FUNCTION_BLOCK FB3_HmiTF1800_UserlevelManagement
VAR_INPUT
	
	bLoginPB 					: BOOL;
	bLogoutPB 					: BOOL;
	iLoginNameId 				: REFERENCE TO INT; // The LoginName selection in HMI during User Login Pop-up Screen, the choosen user will translated as Array ID No and pass here.
	sPasswordField 				: REFERENCE TO STRING; // Similar to Var In/Out so that i can clear the password if login failed
	
	iUM_SelectedLoginNameId	 	: REFERENCE TO INT;		// User Management - Selected Login Name ID (Array No)

	sUM_CurrentPassword			: REFERENCE TO STRING;	// User Management - Current Password (For password change only)
	sUM_NewPassword				: REFERENCE TO STRING;	// User Management - New Password (For password change or new user registration)
	sUM_ConfirmPassword			: REFERENCE TO STRING;	// User Management - New Password (For password change or new user registration)

	sUM_NewUserLoginName		: REFERENCE TO STRING;	// User Management - New User Login Name
	sUM_NewUserGroupId			: REFERENCE TO INT;		// User Management - Select from UserGroupList

	sUM_NewUserOperatorIdentifier	: REFERENCE TO STRING;
	sUM_NewUserActorType			: REFERENCE TO eActor;
	sUM_NewUserLastName				: REFERENCE TO STRING;
	sUM_NewUserFirstName			: REFERENCE TO STRING;
//	sUM_NewUserGroupName			: REFERENCE TO WSTRING; // Generated by reference eto sUM_NewUserGroupId
	
	bUM_CreatePB				: BOOL;		// User Management - Button for New User creation
	bUM_EditPB					: BOOL;		// User Management - Button for Edit User
	bUM_DeletePB				: BOOL;		// User Management - Button for Delete User
	bUM_EnablePB				: BOOL; 	// to Enable selected User
	bUM_DisablePB				: BOOL; 	// to Temporary Disable selected User
	bUM_ConfirmPB				: BOOL;		// for Edit, Delete and Disable used. click to save
	bUM_ReturnPB				: BOOL;		// for Edit, Delete and Disable used, click to return without save.
		
END_VAR
VAR_OUTPUT
	dsHmiUserStatus_Active		: DS_HmiUserStatus;
	dsHmiUserStatus_Login		: DS_HmiUserStatus;
	dsHmiUserStatus_Logout		: DS_HmiUserStatus;
	
//	iActiveUserGroupId			: INT;
//	sActiveLoginName			: STRING;
	
//	sActiveOperatorIdentifier	: STRING;
//	eActiveActorType			: eActor;
//	sActiveLastName				: STRING;
//	sActiveFirstName			: STRING;
	wsActiveUserGroupName		: WSTRING;
	sMessage					: STRING;
	
END_VAR
VAR
	tsLocalSystemTimeStruct		: TIMESTRUCT;
	dsHmiUserStatus_Empty		: DS_HmiUserStatus;

	ARsUserGroup 				: ARRAY [0..5] OF WSTRING;	// Default UserGroup - Must Matched with HMI UserGroup Naming
	
	bLoginPBRE		: R_TRIG;
	bLogoutPBRE		: R_TRIG;
	bUM_CreatePBRE	: R_TRIG;
	bUM_EditPBRE	: R_TRIG;
	bUM_DeletePBRE	: R_TRIG;
	bUM_DisablePBRE	: R_TRIG;
	iCase: INT;
	sMessageDelayTimer: TON;
	iFL: INT;
	bDuplicatedLoginName: BOOL;
	bDuplicatedOperatorId: BOOL;
	bUserDBMax: BOOL;
	iUserDBVacantField: INT;
	bUM_ConfirmPBRE: R_TRIG;
	bUM_ReturnPBRE: R_TRIG;
	btest: BOOL;
	bUM_EnablePBRE: R_TRIG;
	tLoginActivatedTimer: TON;
	tLogoutActivatedTimer: TON;
	ntGetTime: NT_GetTime;
	t1s: TON;
END_VAR
	
VAR PERSISTENT
	dsHmiUserReg 			: DS_HmiUserReg;
END_VAR

t1s(IN:=NOT t1s.Q , PT:=T#0.5S , Q=> , ET=> );

// Get System Time
ntGetTime(	NETID:='' , START:=t1s.Q , TMOUT:= T#5S, TIMESTR=> tsLocalSystemTimeStruct);

tsLocalSystemTimeStruct.wYear;
tsLocalSystemTimeStruct.wMonth;
tsLocalSystemTimeStruct.wDay;
tsLocalSystemTimeStruct.wHour;
tsLocalSystemTimeStruct.wMinute;
tsLocalSystemTimeStruct.wSecond;
tsLocalSystemTimeStruct.wMilliseconds;
tsLocalSystemTimeStruct.wDayOfWeek;


// Default UserGroup - Must Matched with HMI UserGroup Naming
ARsUserGroup[0]			:= 	STRING_TO_WSTRING('GUEST');
ARsUserGroup[1]			:= 	STRING_TO_WSTRING('OPERATOR');
ARsUserGroup[2]			:=	STRING_TO_WSTRING('TECHNICIAN');
ARsUserGroup[3]			:=	STRING_TO_WSTRING('ENGINEER');
ARsUserGroup[4]			:=	STRING_TO_WSTRING('ADMIN');
ARsUserGroup[5]			:=	STRING_TO_WSTRING('JKS');
//ARsUserGroup[6]			:=	STRING_TO_WSTRING('');
//ARsUserGroup[7]			:=	STRING_TO_WSTRING('');	

// Default SuperAdmin
dsHmiUserReg.ARbUserStatus[dsHmiUserReg.iQtyUserReg+1]			:= 	TRUE		;
dsHmiUserReg.AReActorType[dsHmiUserReg.iQtyUserReg+1]			:= 	0			; //Human
dsHmiUserReg.ARiUserGroupID[dsHmiUserReg.iQtyUserReg+1]			:= 	5			; //Highest level - JKS Admin
dsHmiUserReg.ARsFirstName[dsHmiUserReg.iQtyUserReg+1]			:= 	'Machine'	;
dsHmiUserReg.ARsLastName[dsHmiUserReg.iQtyUserReg+1]			:= 	'Maker'		;
dsHmiUserReg.ARsLoginName[dsHmiUserReg.iQtyUserReg+1]			:= 	'SoftwareManager'	;
dsHmiUserReg.ARsOperatorIdentifier[dsHmiUserReg.iQtyUserReg+1]	:= 	'Software Manager'	;
dsHmiUserReg.ARsPw[dsHmiUserReg.iQtyUserReg+1]					:= 	'7189'	;
dsHmiUserReg.ARwsUserGroupName[dsHmiUserReg.iQtyUserReg+1]		:= 	ARsUserGroup[5]	;


// R_TRIG
bLoginPBRE		(CLK:=bLoginPB , 		Q=> );
bLogoutPBRE		(CLK:=bLogoutPB , 		Q=> );

bUM_CreatePBRE	(CLK:=bUM_CreatePB , 	Q=> );
bUM_EditPBRE	(CLK:=bUM_EditPB , 		Q=> );
bUM_DeletePBRE	(CLK:=bUM_DeletePB , 	Q=> );
bUM_EnablePBRE	(CLK:=bUM_EnablePB , 	Q=> );
bUM_DisablePBRE	(CLK:=bUM_DisablePB , 	Q=> );
bUM_ConfirmPBRE	(CLK:=bUM_ConfirmPB , 	Q=> );
bUM_ReturnPBRE	(CLK:=bUM_ReturnPB , 	Q=> );


// Delay off
tLoginActivatedTimer(IN:=dsHmiUserStatus_Login.bActivatedFlag , PT:=T#1S , Q=> , ET=> );
IF tLoginActivatedTimer.Q THEN
	dsHmiUserStatus_Login.bActivatedFlag := FALSE;
END_IF

tLogoutActivatedTimer(IN:=dsHmiUserStatus_Logout.bActivatedFlag , PT:=T#1S , Q=> , ET=> );
IF tLogoutActivatedTimer.Q THEN
	dsHmiUserStatus_Logout.bActivatedFlag := FALSE;
END_IF



// Action 

	IF iCase = 0 THEN
		
		IF 	bLoginPBRE.Q AND iLoginNameId > 0 AND iLoginNameId <= dsHmiUserReg.iQtyUserReg +1 AND sPasswordField <> '' THEN
			iCase := 11; // Login 
			
		ELSIF bLogoutPBRE.Q THEN
			iCase := 21; //	Logout
			
		ELSIF bUM_CreatePBRE.Q AND dsHmiUserStatus_Login.sUserGroupId >= 4 THEN
			iCase := 31; //	User Management -> New User Creation
			
		ELSIF bUM_EditPBRE.Q AND dsHmiUserStatus_Login.sUserGroupId >= 4 AND iUM_SelectedLoginNameId > 0 AND iUM_SelectedLoginNameId <= dsHmiUserReg.iQtyUserReg +1 THEN
			iCase := 41; //	User Management -> Edit User
			
		ELSIF bUM_DeletePBRE.Q AND dsHmiUserStatus_Login.sUserGroupId >= 4 AND iUM_SelectedLoginNameId > 0 AND iUM_SelectedLoginNameId <= dsHmiUserReg.iQtyUserReg +1 
		AND dsHmiUserReg.ARsLoginName[iUM_SelectedLoginNameId] <> dsHmiUserStatus_Login.sLoginName THEN
			iCase := 51; //	User Management -> Delete User
			
		ELSIF (bUM_EnablePBRE.Q OR bUM_DisablePBRE.Q)AND dsHmiUserStatus_Login.sUserGroupId >= 4 AND iUM_SelectedLoginNameId > 0 AND iUM_SelectedLoginNameId <= dsHmiUserReg.iQtyUserReg +1 THEN
			iCase := 61; //	User Management -> Enable or Temporary Disable selected User

		ELSIF (bUM_DeletePBRE.Q) AND dsHmiUserReg.ARsLoginName[iUM_SelectedLoginNameId] = dsHmiUserStatus_Login.sLoginName THEN
				sMessage := 'Signed in user cannot be delete, please sign in another administrator user before deletion';
					
		ELSIF (bUM_CreatePBRE.Q OR bUM_EditPBRE.Q OR bUM_DeletePBRE.Q OR bUM_EnablePBRE.Q OR bUM_DisablePBRE.Q ) AND dsHmiUserStatus_Login.sUserGroupId <= 4  THEN
				sMessage := 'You do not have permission to perform the task, please contact administrator.';
					
		ELSIF (bUM_EditPBRE.Q OR bUM_DeletePBRE.Q OR bUM_EnablePBRE.Q OR bUM_DisablePBRE.Q ) AND iUM_SelectedLoginNameId = 0 THEN
				sMessage := 'Please select user';
					
		ELSIF (bUM_EditPBRE.Q OR bUM_DeletePBRE.Q OR bUM_EnablePBRE.Q OR bUM_DisablePBRE.Q ) AND iUM_SelectedLoginNameId > dsHmiUserReg.iQtyUserReg +1 THEN
				sMessage := 'Selected user out of user database range';
					
		ELSIF bLoginPBRE.Q AND (iLoginNameId = 0 OR sPasswordField = '' ) THEN
				sMessage := 'Please select user and enter password to login';
					
		ELSIF bLoginPBRE.Q AND iLoginNameId > dsHmiUserReg.iQtyUserReg +1 THEN
				sMessage := 'Selected login user out of user database range';
					
		END_IF
		
	END_IF



CASE iCase OF
	
	0: ;// Idling;

	8: // Clear new user registration field and return

		sUM_CurrentPassword 			:= '' ;
		sUM_NewPassword 				:= '' ;
		sUM_ConfirmPassword 			:= '' ; 
		sUM_NewUserLoginName 			:= '' ; 
		sUM_NewUserGroupId				:= 0 ;	
		sUM_NewUserOperatorIdentifier	:= '' ;
		sUM_NewUserActorType			:= 0 ; 
		sUM_NewUserLastName				:= '' ;
		sUM_NewUserFirstName			:= '' ;
		
		iUM_SelectedLoginNameId			:= 0;
		
		iCase := 0; // Return		
	
	9: // Clear Active Field and return
	
		dsHmiUserStatus_Logout := dsHmiUserStatus_Active;
		IF dsHmiUserStatus_Logout.sLoginName <> '' THEN
			dsHmiUserStatus_Logout.bActivatedFlag 	:= TRUE;
			dsHmiUserStatus_Logout.tsDateTime 		:= tsLocalSystemTimeStruct;
		END_IF

		sPasswordField 			:= 		'';
		dsHmiUserStatus_Active 	:= 		dsHmiUserStatus_Empty;
		wsActiveUserGroupName 	:= 		TO_WSTRING('');

		iCase := 0; //Return



	11: // Login 
	
		IF dsHmiUserReg.ARsPw[iLoginNameId] = sPasswordField AND dsHmiUserReg.ARbUserStatus[iLoginNameId] THEN
				
				// if detected with existing login user and it relogin with another user, this section will action
				IF dsHmiUserStatus_Active.sLoginName <> '' THEN
					dsHmiUserStatus_Logout := dsHmiUserStatus_Active;
					dsHmiUserStatus_Logout.bActivatedFlag := TRUE;
					dsHmiUserStatus_Logout.tsDateTime := tsLocalSystemTimeStruct;
				END_IF


				sPasswordField 				:= 		'';
				
				dsHmiUserStatus_Active.bActivatedFlag		:= 		TRUE;
				dsHmiUserStatus_Active.sOperatorIdentifier 	:= 		dsHmiUserReg.ARsOperatorIdentifier[iLoginNameId];	// Celestica Requirement
				dsHmiUserStatus_Active.eActorType			:=		dsHmiUserReg.AReActorType[iLoginNameId];			// Celestica Requirement
				dsHmiUserStatus_Active.sULastName			:=		dsHmiUserReg.ARsLastName[iLoginNameId];
				dsHmiUserStatus_Active.sFirstName			:=		dsHmiUserReg.ARsFirstName[iLoginNameId];
				
				dsHmiUserStatus_Active.sLoginName			:=		dsHmiUserReg.ARsLoginName[iLoginNameId];			// Same as Username
	
				dsHmiUserStatus_Active.sUserGroupId			:=		dsHmiUserReg.ARiUserGroupID[iLoginNameId];			// Define in HMI TF1800

				dsHmiUserStatus_Active.tsDateTime			:=		tsLocalSystemTimeStruct;
				wsActiveUserGroupName 						:= 		dsHmiUserReg.ARwsUserGroupName[iLoginNameId];
				
	
				dsHmiUserStatus_Login := dsHmiUserStatus_Active;
				dsHmiUserStatus_Login.bActivatedFlag := TRUE;
				dsHmiUserStatus_Login.tsDateTime := tsLocalSystemTimeStruct;
				
				sMessage := 'Welcome!';
				sMessage := concat(sMessage,' ');
				sMessage := concat(sMessage,dsHmiUserStatus_Active.sFirstName);
				sMessage := concat(sMessage,' ');
				sMessage := concat(sMessage,dsHmiUserStatus_Active.sULastName);
				sMessage := concat(sMessage,' (');
				sMessage := concat(sMessage,dsHmiUserStatus_Active.sLoginName);
				sMessage := concat(sMessage,')');
		
				iCase := 0;	//Return
						
		ELSIF NOT dsHmiUserReg.ARbUserStatus[iLoginNameId] THEN
				sMessage := 'Selected user has been DISABLE, please contact administrator.';
				iCase := 9; // Clear Active Field and return
			
		
		ELSE
				sMessage := 'Invalid password';
				iCase := 9; // Clear Active Field and return
		
		END_IF
				
		
	
	21: // Logout 
		
				sMessage := 'You have been successfully logged out.';	
				iCase := 9; // Clear Active Field and return 
		
	
	31: // User Management -> New User Creation 
	
		IF sUM_NewPassword 					<> '' 
		AND sUM_ConfirmPassword 			<> '' 
	//	AND sUM_NewUserLoginName 			<> '' 
		AND sUM_NewUserGroupId				<> 0 AND sUM_NewUserGroupId <= 4	// Doesnt need for another JKS User (5)
	//	AND sUM_NewUserOperatorIdentifier	<> ''
	//	AND sUM_NewUserActorType			<= 2 AND sUM_NewUserActorType >= 0
		AND sUM_NewUserLastName				<> ''
		AND sUM_NewUserFirstName			<> ''

		THEN
			
			// Check Duplicated Login Name
				bDuplicatedLoginName := FALSE;
				
				FOR iFL := 1 TO dsHmiUserReg.iQtyUserReg DO
					IF sUM_NewUserLoginName = dsHmiUserReg.ARsLoginName[iFL] THEN
						bDuplicatedLoginName := TRUE;
						EXIT;
					END_IF
				;
				END_FOR

			// Check Duplicated Operator Identifier
				bDuplicatedOperatorId := FALSE;
				
				FOR iFL := 1 TO dsHmiUserReg.iQtyUserReg DO
					IF sUM_NewUserOperatorIdentifier = dsHmiUserReg.ARsOperatorIdentifier[iFL] THEN
						bDuplicatedOperatorId := TRUE;
						EXIT;
					END_IF
				;
				END_FOR

			// Check User Database Limit
				bUserDBMax := TRUE;
				iUserDBVacantField := 0;
				
				FOR iFL := 1 TO dsHmiUserReg.iQtyUserReg DO
					IF dsHmiUserReg.ARsLoginName[iFL] = '' THEN
						iUserDBVacantField := iFL;
						bUserDBMax := FALSE;
						EXIT;
					END_IF
				;
				END_FOR


			IF sUM_NewPassword <> sUM_ConfirmPassword THEN
				
				sMessage := 'Your new password and confirmation password mismatched';	
				sUM_ConfirmPassword := '';
				iCase := 0;

			ELSIF bDuplicatedLoginName THEN
							
				sMessage := 'Login Name already exists, please try with another one ';	
				sUM_NewUserLoginName 	:= '';
				sUM_NewPassword			:= '';
				sUM_ConfirmPassword 	:= '';
				iCase 					:= 0;

//			ELSIF bDuplicatedOperatorId THEN
							
//				sMessage := 'Operator Indentifier already exists, please try with another one ';	
//				sUM_NewUserOperatorIdentifier 	:= '';
//				sUM_NewPassword					:= '';
//				sUM_ConfirmPassword 			:= '';
//				iCase 							:= 0;
				
			ELSIF bUserDBMax THEN
							
				sMessage 	:= 'User Registration Limit Reached. Please delete at least one user to proceed the registration again ';	
				iCase 		:= 8; // Clear new user registration field and return
				
			ELSE
				
				
							
			//	dsHmiUserReg.ARsOperatorIdentifier[iUserDBVacantField] 	:= sUM_NewUserOperatorIdentifier;	// Celestica Requirement
			//	dsHmiUserReg.AReActorType[iUserDBVacantField]			:= sUM_NewUserActorType;			// Celestica Requirement
				dsHmiUserReg.ARsLastName[iUserDBVacantField]			:= sUM_NewUserLastName;
				dsHmiUserReg.ARsFirstName[iUserDBVacantField]			:= sUM_NewUserFirstName;
				dsHmiUserReg.ARsLoginName[iUserDBVacantField]			:= sUM_NewUserLoginName;			// Same as Username
				dsHmiUserReg.ARbUserStatus[iUserDBVacantField]			:= TRUE;							// 0 = Deactivated/Disable, 1 = Active User
				
				dsHmiUserReg.ARiUserGroupID[iUserDBVacantField]			:= sUM_NewUserGroupId;				// Define in HMI TF1800
				dsHmiUserReg.ARwsUserGroupName[iUserDBVacantField]		:= ARsUserGroup[sUM_NewUserGroupId];// Define in HMI TF1800
				dsHmiUserReg.ARsPw[iUserDBVacantField]					:= sUM_NewPassword;		

				sMessage := 'User is added successfully. Please go to Login page to proceed';	
				iCase := 8; // Clear new user registration field and return
					
			END_IF
			
		
		ELSE
			
			sMessage := 'Your registration is Incomplete';	
			iCase := 0; //RETURN
		END_IF
	
		
	41: // User Management -> Edit User 

		sUM_NewUserOperatorIdentifier := dsHmiUserReg.ARsOperatorIdentifier[iUM_SelectedLoginNameId];	// Celestica Requirement
		sUM_NewUserActorType := dsHmiUserReg.AReActorType[iUM_SelectedLoginNameId];						// Celestica Requirement
		sUM_NewUserLastName := dsHmiUserReg.ARsLastName[iUM_SelectedLoginNameId];
		sUM_NewUserFirstName := dsHmiUserReg.ARsFirstName[iUM_SelectedLoginNameId];
		sUM_NewUserLoginName := dsHmiUserReg.ARsLoginName[iUM_SelectedLoginNameId];						// Same as Username
		
		sUM_NewUserGroupId := dsHmiUserReg.ARiUserGroupID[iUM_SelectedLoginNameId];						// Define in HMI TF1800

		sUM_CurrentPassword := '';//dsHmiUserReg.ARsPw[iUM_SelectedLoginNameId];		
		sUM_NewPassword 	:= '';//dsHmiUserReg.ARsPw[iUM_SelectedLoginNameId];		
		sUM_ConfirmPassword := '';//dsHmiUserReg.ARsPw[iUM_SelectedLoginNameId];		
		
		iCase := 42;

	42: // User Management -> Edit User => Waiting Confirmation
	
		sMessage := 'Are you sure you want to MODIFY selected user?';	
	
		IF bUM_ConfirmPBRE.Q THEN
					
			IF sUM_CurrentPassword <> dsHmiUserReg.ARsPw[iUM_SelectedLoginNameId] THEN
					
				sMessage := 'Invalid Current Password';
				iUM_SelectedLoginNameId := 0;	
				iCase := 8; // Clear and return
			
			ELSIF sUM_NewPassword <> sUM_ConfirmPassword THEN	
			
					
				sMessage := 'Your new password and confirmation password mismatched';
				iUM_SelectedLoginNameId := 0;	
				iCase := 8; // Clear and return
			
			ELSE
				dsHmiUserReg.ARsOperatorIdentifier[iUM_SelectedLoginNameId] 	:= sUM_NewUserOperatorIdentifier;	// Celestica Requirement
				dsHmiUserReg.AReActorType[iUM_SelectedLoginNameId]				:= sUM_NewUserActorType;			// Celestica Requirement
				dsHmiUserReg.ARsLastName[iUM_SelectedLoginNameId]				:= sUM_NewUserLastName;
				dsHmiUserReg.ARsFirstName[iUM_SelectedLoginNameId]				:= sUM_NewUserFirstName;
				dsHmiUserReg.ARsLoginName[iUM_SelectedLoginNameId]				:= sUM_NewUserLoginName;			// Same as Username
				//dsHmiUserReg.ARbUserStatus[iUM_SelectedLoginNameId]			:= TRUE;							// 0 = Deactivated/Disable, 1 = Active User
				
				dsHmiUserReg.ARiUserGroupID[iUM_SelectedLoginNameId]			:= sUM_NewUserGroupId;				// Define in HMI TF1800
				dsHmiUserReg.ARwsUserGroupName[iUM_SelectedLoginNameId]			:= ARsUserGroup[sUM_NewUserGroupId];// Define in HMI TF1800
				
				IF sUM_NewPassword <> '' THEN
					dsHmiUserReg.ARsPw[iUM_SelectedLoginNameId]						:= sUM_NewPassword;		// It will only update the password if the New and Confirm password filled accurately.
				END_IF
				
				sMessage := 'User Info is Updated successfully. Please go to Login page to proceed';	
				iUM_SelectedLoginNameId := 0;	
				iCase := 8; // Clear new user registration field and return
	
			END_IF
				
		ELSIF bUM_ReturnPBRE.Q THEN

			sMessage := 'Returned';	
			iUM_SelectedLoginNameId := 0;	
			iCase := 8; // Clear and return

		END_IF		
	51: // User Management -> Delete User 
	
		sMessage := 'Are you sure you want to DELETE selected user?';	
	
		IF bUM_ConfirmPBRE.Q THEN 
					
			dsHmiUserReg.ARsOperatorIdentifier[iUM_SelectedLoginNameId]		:= '';				// Celestica Requirement
			dsHmiUserReg.AReActorType[iUM_SelectedLoginNameId]				:= 0;				// Celestica Requirement
			dsHmiUserReg.ARsLastName[iUM_SelectedLoginNameId]				:= '';
			dsHmiUserReg.ARsFirstName[iUM_SelectedLoginNameId]				:= '';
			dsHmiUserReg.ARsLoginName[iUM_SelectedLoginNameId]				:= '';				// Same as Username
			dsHmiUserReg.ARbUserStatus[iUM_SelectedLoginNameId]				:= FALSE;			// 0 = Deactivated/Disable, 1 = Active User
			
			dsHmiUserReg.ARiUserGroupID[iUM_SelectedLoginNameId]			:= 0;				// Define in HMI TF1800
			dsHmiUserReg.ARwsUserGroupName[iUM_SelectedLoginNameId]			:= TO_WSTRING('');	// Define in HMI TF1800
			dsHmiUserReg.ARsPw[iUM_SelectedLoginNameId]						:= '';					

			sMessage := 'Selected user has been DELETED.';
			iUM_SelectedLoginNameId := 0;	
			iCase := 0;
		
		ELSIF bUM_ReturnPBRE.Q THEN

			sMessage := 'Returned';	
			iUM_SelectedLoginNameId := 0;	
			iCase := 0;

		END_IF

	61: // User Management -> Temporary Disable selected User 
	
		IF bUM_EnablePBRE.Q THEN
			 sMessage := 'Are you sure you want to ENABLE selected user?';	

		ELSIF bUM_DisablePBRE.Q THEN
			 sMessage := 'Are you sure you want to DISABLE selected user?';	
		END_IF
	

	
		IF bUM_ConfirmPBRE.Q AND sMessage = 'Are you sure you want to ENABLE selected user?' THEN 
					
			dsHmiUserReg.ARbUserStatus[iUM_SelectedLoginNameId]				:= TRUE;			// 0 = Deactivated/Disable, 1 = Active User			
			sMessage := 'Selected user has been ENABLE.';	
			iUM_SelectedLoginNameId := 0;	
			iCase := 0;
		
		ELSIF bUM_ConfirmPBRE.Q AND sMessage = 'Are you sure you want to DISABLE selected user?' THEN 			
					
			dsHmiUserReg.ARbUserStatus[iUM_SelectedLoginNameId]				:= FALSE;			// 0 = Deactivated/Disable, 1 = Active User			
			sMessage := 'Selected user has been DISABLE.';	
			iUM_SelectedLoginNameId := 0;	
			iCase := 0;
		
		ELSIF bUM_ReturnPBRE.Q THEN

			sMessage := 'Returned';	
			iUM_SelectedLoginNameId := 0;	
			iCase := 0;

		END_IF

END_CASE



// Clear Message after x period of time
	
	sMessageDelayTimer(IN:=sMessage <> '' AND iCase <> 42 AND iCase <> 51 AND iCase <> 61 , PT:=T#3S , Q=> , ET=> );
	IF sMessageDelayTimer.Q THEN
		sMessage := '';
	END_IF

END_FUNCTION_BLOCK

(* stored: Version 1.1.0.1, ProductVersion 3.1.4024.12
   POU FB3_HmiTF1800_UserlevelManagement: Id {ee5f859a-e9ec-4d96-b04e-63d1d0ad6c10}, SpecialFunc None *)
